TYPE DUT :
STRUCT
	b : BOOL;
	n : BOOL;
	m : BOOL;
END_STRUCT
END_TYPE

(* stored: Version 1.1.0.1, ProductVersion 3.1.4024.12
   DUT DUT: Id {91eee736-4b0e-4b17-a608-2ba691a0e60a} *)
